TYPE Ethercat_AlarmsWarningToCLC :
STRUCT
	Communication_Alarms : BOOL; 
	Battery_Alarms : BOOL;
	Warnings: BOOL;
	Faults: BOOL;
	reservebit1 : BOOL;
	reservebit2 : BOOL;
	reservebit3 : BOOL;
	reservebit4 : BOOL;

END_STRUCT
END_TYPE

(* stored: Version 1.1.0.1, ProductVersion 3.1.4024.11
   DUT Ethercat_AlarmsWarningToCLC: Id {a7f74e27-b9b5-4af4-a36e-68018fe96641} *)
